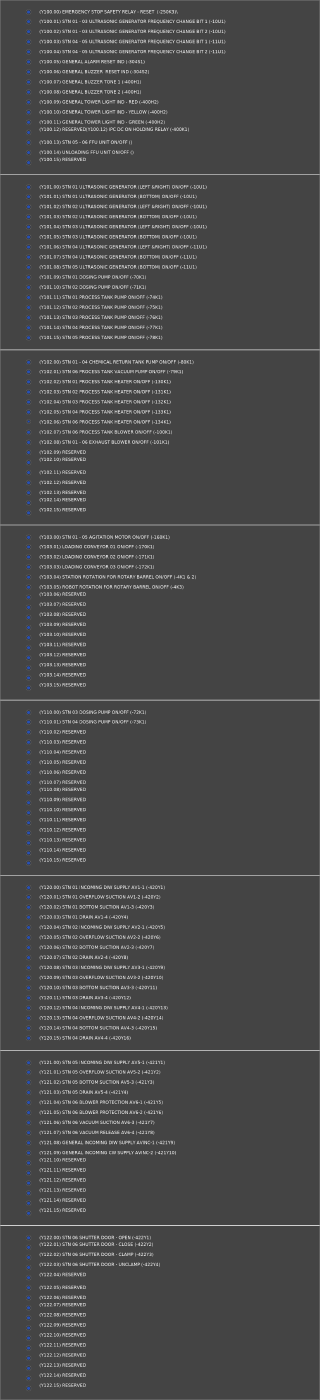
VISUALIZATION Popup_IOoutput  // 733x3198
    Rectangle (0,0 733x398)
    Label (87,15 625x24), "(Y100.00) EMERGENCY STOP SAFETY RELAY - RESET (-250K3)\"
    Label (87,37 625x24), "(Y100.01) STN 01 - 03 ULTRASONIC GENERATOR FREQUENCY CHANGE BIT 1 (-10U1)"
    Label (87,83 625x24), "(Y100.03) STN 04 - 05 ULTRASONIC GENERATOR FREQUENCY CHANGE BIT 1 (-11U1)"
    Label (87,60 625x24), "(Y100.02) STN 01 - 03 ULTRASONIC GENERATOR FREQUENCY CHANGE BIT 2 (-10U1)"
    Label (87,175 625x24), "(Y100.07) GENERAL BUZZER TONE 1 (-400H1)"
    Label (87,106 625x24), "(Y100.04) STN 04 - 05 ULTRASONIC GENERATOR FREQUENCY CHANGE BIT 2 (-11U1)"
    Label (87,129 625x24), "(Y100.05) GENERAL ALARM RESET IND (-304S1)"
    Label (87,152 625x24), "(Y100.06) GENERAL BUZZER RESET IND (-304S2)"
    Label (87,359 625x24), "(Y100.15) RESERVED"
    Label (87,198 625x24), "(Y100.08) GENERAL BUZZER TONE 2 (-400H1)"
    Label (87,221 625x24), "(Y100.09) GENERAL TOWER LIGHT IND - RED (-400H2)"
    Label (87,267 625x24), "(Y100.11) GENERAL TOWER LIGHT IND - GREEN (-400H2)"
    Label (87,244 625x24), "(Y100.10) GENERAL TOWER LIGHT IND - YELLOW (-400H2)"
    Label (87,290 625x24), "(Y100.12) RESERVED(Y100.12) IPC DC ON HOLDING RELAY (-400K1)"
    Label (87,313 625x24), "(Y100.13) STN 05 - 06 FFU UNIT ON/OFF ()"
    Label (87,336 625x24), "(Y100.14) UNLOADING FFU UNIT ON/OFF ()"
    Rectangle (0,400 733x398)
    Label (87,415 625x24), "(Y101.00) STN 01 ULTRASONIC GENERATOR (LEFT &RIGHT) ON/OFF (-10U1)"
    Label (87,437 625x24), "(Y101.01) STN 01 ULTRASONIC GENERATOR (BOTTOM) ON/OFF (-10U1)"
    Label (87,483 625x24), "(Y101.03) STN 02 ULTRASONIC GENERATOR (BOTTOM) ON/OFF (-10U1)"
    Label (87,460 625x24), "(Y101.02) STN 02 ULTRASONIC GENERATOR (LEFT &RIGHT) ON/OFF (-10U1)"
    Label (87,575 625x24), "(Y101.07) STN 04 ULTRASONIC GENERATOR (BOTTOM) ON/OFF (-11U1)"
    Label (87,506 625x24), "(Y101.04) STN 03 ULTRASONIC GENERATOR (LEFT &RIGHT) ON/OFF (-10U1)"
    Label (87,529 625x24), "(Y101.05) STN 03 ULTRASONIC GENERATOR (BOTTOM) ON/OFF (-10U1)"
    Label (87,552 625x24), "(Y101.06) STN 04 ULTRASONIC GENERATOR (LEFT &RIGHT) ON/OFF (-11U1)"
    Label (87,759 625x24), "(Y101.15) STN 05 PROCESS TANK PUMP ON/OFF (-78K1)"
    Label (87,598 625x24), "(Y101.08) STN 05 ULTRASONIC GENERATOR (BOTTOM) ON/OFF (-11U1)"
    Label (87,621 625x24), "(Y101.09) STN 01 DOSING PUMP ON/OFF (-70K1)"
    Label (87,667 625x24), "(Y101.11) STN 01 PROCESS TANK PUMP ON/OFF (-74K1)"
    Label (87,644 625x24), "(Y101.10) STN 02 DOSING PUMP ON/OFF (-71K1)"
    Label (87,690 625x24), "(Y101.12) STN 02 PROCESS TANK PUMP ON/OFF (-75K1)"
    Label (87,713 625x24), "(Y101.13) STN 03 PROCESS TANK PUMP ON/OFF (-76K1)"
    Label (87,736 625x24), "(Y101.14) STN 04 PROCESS TANK PUMP ON/OFF (-77K1)"
    Rectangle (0,800 733x398)
    Label (87,815 625x24), "(Y102.00) STN 01 - 04 CHEMICAL RETURN TANK PUMP ON/OFF (-80K1)"
    Label (87,837 625x24), "(Y102.01) STN 06 PROCESS TANK VACUUM PUMP ON/OFF (-79K1)"
    Label (87,883 625x24), "(Y102.03) STN 02 PROCESS TANK HEATER ON/OFF (-131K1)"
    Label (87,860 625x24), "(Y102.02) STN 01 PROCESS TANK HEATER ON/OFF (-130K1)"
    Label (87,975 625x24), "(Y102.07) STN 06 PROCESS TANK BLOWER ON/OFF (-100K1)"
    Label (87,906 625x24), "(Y102.04) STN 03 PROCESS TANK HEATER ON/OFF (-132K1)"
    Label (87,929 625x24), "(Y102.05) STN 04 PROCESS TANK HEATER ON/OFF (-133K1)"
    Label (87,952 625x24), "(Y102.06) STN 06 PROCESS TANK HEATER ON/OFF (-134K1)"
    Label (87,1159 625x24), "(Y102.15) RESERVED"
    Label (87,998 625x24), "(Y102.08) STN 01 - 06 EXHAUST BLOWER ON/OFF (-101K1)"
    Label (87,1021 625x24), "(Y102.09) RESERVED"
    Label (87,1067 625x24), "(Y102.11) RESERVED"
    Label (87,1044 625x24), "(Y102.10) RESERVED"
    Label (87,1090 625x24), "(Y102.12) RESERVED"
    Label (87,1113 625x24), "(Y102.13) RESERVED"
    Label (87,1136 625x24), "(Y102.14) RESERVED"
    Rectangle (0,1600 733x398)
    Label (87,1615 625x24), "(Y110.00) STN 03 DOSING PUMP ON/OFF (-72K1)"
    Label (87,1637 625x24), "(Y110.01) STN 04 DOSING PUMP ON/OFF (-73K1)"
    Label (87,1683 625x24), "(Y110.03) RESERVED"
    Label (87,1660 625x24), "(Y110.02) RESERVED"
    Label (87,1775 625x24), "(Y110.07) RESERVED"
    Label (87,1706 625x24), "(Y110.04) RESERVED"
    Label (87,1729 625x24), "(Y110.05) RESERVED"
    Label (87,1752 625x24), "(Y110.06) RESERVED"
    Label (87,1959 625x24), "(Y110.15) RESERVED"
    Label (87,1798 625x24), "(Y110.08) RESERVED"
    Label (87,1821 625x24), "(Y110.09) RESERVED"
    Label (87,1867 625x24), "(Y110.11) RESERVED"
    Label (87,1844 625x24), "(Y110.10) RESERVED"
    Label (87,1890 625x24), "(Y110.12) RESERVED"
    Label (87,1913 625x24), "(Y110.13) RESERVED"
    Label (87,1936 625x24), "(Y110.14) RESERVED"
    Rectangle (0,1200 733x398)
    Label (87,1215 625x24), "(Y103.00) STN 01 - 05 AGITATION MOTOR ON/OFF (-160K1)"
    Label (87,1237 625x24), "(Y103.01) LOADING CONVEYOR 01 ON/OFF (-170K1)"
    Label (87,1283 625x24), "(Y103.03) LOADING CONVEYOR 03 ON/OFF (-172K1)"
    Label (87,1260 625x24), "(Y103.02) LOADING CONVEYOR 02 ON/OFF (-171K1)"
    Label (87,1375 625x24), "(Y103.07) RESERVED"
    Label (87,1306 625x24), "(Y103.04) STATION ROTATION FOR ROTARY BARREL ON/OFF (-4K1 & 2)"
    Label (87,1329 625x24), "(Y103.05) ROBOT ROTATION FOR ROTARY BARREL ON/OFF (-4K3)"
    Label (87,1352 625x24), "(Y103.06) RESERVED"
    Label (87,1559 625x24), "(Y103.15) RESERVED"
    Label (87,1398 625x24), "(Y103.08) RESERVED"
    Label (87,1421 625x24), "(Y103.09) RESERVED"
    Label (87,1467 625x24), "(Y103.11) RESERVED"
    Label (87,1444 625x24), "(Y103.10) RESERVED"
    Label (87,1490 625x24), "(Y103.12) RESERVED"
    Label (87,1513 625x24), "(Y103.13) RESERVED"
    Label (87,1536 625x24), "(Y103.14) RESERVED"
    Rectangle (0,2000 733x398)
    Label (87,2015 625x24), "(Y120.00) STN 01 INCOMING DIW SUPPLY AV1-1 (-420Y1)"
    Label (87,2037 625x24), "(Y120.01) STN 01 OVERFLOW SUCTION AV1-2 (-420Y2)"
    Label (87,2083 625x24), "(Y120.03) STN 01 DRAIN AV1-4 (-420Y4)"
    Label (87,2060 625x24), "(Y120.02) STN 01 BOTTOM SUCTION AV1-3 (-420Y3)"
    Label (87,2175 625x24), "(Y120.07) STN 02 DRAIN AV2-4 (-420Y8)"
    Label (87,2106 625x24), "(Y120.04) STN 02 INCOMING DIW SUPPLY AV2-1 (-420Y5)"
    Label (87,2129 625x24), "(Y120.05) STN 02 OVERFLOW SUCTION AV2-2 (-420Y6)"
    Label (87,2152 625x24), "(Y120.06) STN 02 BOTTOM SUCTION AV2-3 (-420Y7)"
    Label (87,2359 625x24), "(Y120.15) STN 04 DRAIN AV4-4 (-420Y16)"
    Label (87,2198 625x24), "(Y120.08) STN 03 INCOMING DIW SUPPLY AV3-1 (-420Y9)"
    Label (87,2221 625x24), "(Y120.09) STN 03 OVERFLOW SUCTION AV3-2 (-420Y10)"
    Label (87,2267 625x24), "(Y120.11) STN 03 DRAIN AV3-4 (-420Y12)"
    Label (87,2244 625x24), "(Y120.10) STN 03 BOTTOM SUCTION AV3-3 (-420Y11)"
    Label (87,2290 625x24), "(Y120.12) STN 04 INCOMING DIW SUPPLY AV4-1 (-420Y13)"
    Label (87,2313 625x24), "(Y120.13) STN 04 OVERFLOW SUCTION AV4-2 (-420Y14)"
    Label (87,2336 625x24), "(Y120.14) STN 04 BOTTOM SUCTION AV4-3 (-420Y15)"
    Rectangle (0,2400 733x398)
    Label (87,2415 625x24), "(Y121.00) STN 05 INCOMING DIW SUPPLY AV5-1 (-421Y1)"
    Label (87,2437 625x24), "(Y121.01) STN 05 OVERFLOW SUCTION AV5-2 (-421Y2)"
    Label (87,2483 625x24), "(Y121.03) STN 05 DRAIN AV5-4 (-421Y4)"
    Label (87,2460 625x24), "(Y121.02) STN 05 BOTTOM SUCTION AV5-3 (-421Y3)"
    Label (87,2575 625x24), "(Y121.07) STN 06 VACUUM RELEASE AV6-4 (-421Y8)"
    Label (87,2506 625x24), "(Y121.04) STN 06 BLOWER PROTECTION AV6-1 (-421Y5)"
    Label (87,2529 625x24), "(Y121.05) STN 06 BLOWER PROTECTION AV6-2 (-421Y6)"
    Label (87,2552 625x24), "(Y121.06) STN 06 VACUUM SUCTION AV6-3 (-421Y7)"
    Label (87,2759 625x24), "(Y121.15) RESERVED"
    Label (87,2598 625x24), "(Y121.08) GENERAL INCOMING DIW SUPPLY AVINC-1 (-421Y9)"
    Label (87,2621 625x24), "(Y121.09) GENERAL INCOMING CW SUPPLY AVINC-2 (-421Y10)"
    Label (87,2667 625x24), "(Y121.11) RESERVED"
    Label (87,2644 625x24), "(Y121.10) RESERVED"
    Label (87,2690 625x24), "(Y121.12) RESERVED"
    Label (87,2713 625x24), "(Y121.13) RESERVED"
    Label (87,2736 625x24), "(Y121.14) RESERVED"
    Rectangle (0,2800 733x398)
    Label (87,2815 625x24), "(Y122.00) STN 06 SHUTTER DOOR - OPEN (-422Y1)"
    Label (87,2837 625x24), "(Y122.01) STN 06 SHUTTER DOOR - CLOSE (-422Y2)"
    Label (87,2883 625x24), "(Y122.03) STN 06 SHUTTER DOOR - UNCLAMP (-422Y4)"
    Label (87,2860 625x24), "(Y122.02) STN 06 SHUTTER DOOR - CLAMP (-422Y3)"
    Label (87,2975 625x24), "(Y122.07) RESERVED"
    Label (87,2906 625x24), "(Y122.04) RESERVED"
    Label (87,2929 625x24), "(Y122.05) RESERVED"
    Label (87,2952 625x24), "(Y122.06) RESERVED"
    Label (87,3159 625x24), "(Y122.15) RESERVED"
    Label (87,2998 625x24), "(Y122.08) RESERVED"
    Label (87,3021 625x24), "(Y122.09) RESERVED"
    Label (87,3067 625x24), "(Y122.11) RESERVED"
    Label (87,3044 625x24), "(Y122.10) RESERVED"
    Label (87,3090 625x24), "(Y122.12) RESERVED"
    Label (87,3113 625x24), "(Y122.13) RESERVED"
    Label (87,3136 625x24), "(Y122.14) RESERVED"
    Lamp1 (58,20 15x15), variable: ARbDO[eY10000_EmergencyStopSafetyRelay_Reset], style: Lamp-Lamp1-Blue
    Lamp1 (58,42 15x15), variable: ARbDO[eY10001_Stn01_03UltrasonicGeneratorFrequencyChangeBit1], style: Lamp-Lamp1-Blue
    Lamp1 (58,88 15x15), variable: ARbDO[eY10004_Stn04_05UltrasonicGeneratorFrequencyChangeBit2], style: Lamp-Lamp1-Blue
    Lamp1 (58,65 15x15), variable: ARbDO[eY10002_Stn01_03UltrasonicGeneratorFrequencyChangeBit2], style: Lamp-Lamp1-Blue
    Lamp1 (58,180 15x15), variable: ARbDO[eY10007_GeneralBuzzerTone1], style: Lamp-Lamp1-Blue
    Lamp1 (58,111 15x15), variable: ARbDI[eX10004_Stn02UltrasonicGeneratorBottom_Alarm], style: Lamp-Lamp1-Blue
    Lamp1 (58,134 15x15), variable: ARbDO[eY10005_GeneralAlarmResetInd], style: Lamp-Lamp1-Blue
    Lamp1 (58,157 15x15), variable: ARbDO[eY10006_GeneralBuzzerResetInd], style: Lamp-Lamp1-Blue
    Lamp1 (58,364 15x15), variable: ARbDO[eY10015_Reserved], style: Lamp-Lamp1-Blue
    Lamp1 (58,203 15x15), variable: ARbDO[eY10008_GeneralBuzzerTone2], style: Lamp-Lamp1-Blue
    Lamp1 (58,226 15x15), variable: ARbDO[eY10009_GeneralTowerLightInd_Red], style: Lamp-Lamp1-Blue
    Lamp1 (58,272 15x15), variable: ARbDO[eY10011_GeneralTowerLightInd_Green], style: Lamp-Lamp1-Blue
    Lamp1 (58,249 15x15), variable: ARbDO[eY10010_GeneralTowerLightInd_Yellow], style: Lamp-Lamp1-Blue
    Lamp1 (58,295 15x15), variable: ARbDO[eY10012_IpcDcOnHoldingRelay], style: Lamp-Lamp1-Blue
    Lamp1 (58,318 15x15), variable: ARbDO[eY10013_Stn05_06FfuUnitOnOff], style: Lamp-Lamp1-Blue
    Lamp1 (58,341 15x15), variable: ARbDO[eY10014_UnloadingFfuUnitOnOff], style: Lamp-Lamp1-Blue
    Lamp1 (58,420 15x15), variable: ARbDO[eY10100_Stn01UltrasonicGeneratorLeftRightOnOff], style: Lamp-Lamp1-Blue
    Lamp1 (58,442 15x15), variable: ARbDO[eY10101_Stn01UltrasonicGeneratorBottomOnOff], style: Lamp-Lamp1-Blue
    Lamp1 (58,488 15x15), variable: ARbDO[eY10103_Stn02UltrasonicGeneratorBottomOnOff], style: Lamp-Lamp1-Blue
    Lamp1 (58,465 15x15), variable: ARbDO[eY10102_Stn02UltrasonicGeneratorLeftRightOnOff], style: Lamp-Lamp1-Blue
    Lamp1 (58,580 15x15), variable: ARbDO[eY10107_Stn04UltrasonicGeneratorBottomOnOff], style: Lamp-Lamp1-Blue
    Lamp1 (58,511 15x15), variable: ARbDO[eY10104_Stn03UltrasonicGeneratorLeftRightOnOff], style: Lamp-Lamp1-Blue
    Lamp1 (58,534 15x15), variable: ARbDO[eY10105_Stn03UltrasonicGeneratorBottomOnOff], style: Lamp-Lamp1-Blue
    Lamp1 (58,557 15x15), variable: ARbDO[eY10106_Stn04UltrasonicGeneratorLeftRightOnOff], style: Lamp-Lamp1-Blue
    Lamp1 (58,764 15x15), variable: ARbDO[eY10115_Stn05ProcessTankPumpOnOff], style: Lamp-Lamp1-Blue
    Lamp1 (58,603 15x15), variable: ARbDO[eY10108_Stn05UltrasonicGeneratorBottomOnOff], style: Lamp-Lamp1-Blue
    Lamp1 (58,626 15x15), variable: ARbDO[eY10109_Stn01DosingPumpOnOff], style: Lamp-Lamp1-Blue
    Lamp1 (58,672 15x15), variable: ARbDO[eY10111_Stn01ProcessTankPumpOnOff], style: Lamp-Lamp1-Blue
    Lamp1 (58,649 15x15), variable: ARbDO[eY10110_Stn02DosingPumpOnOff], style: Lamp-Lamp1-Blue
    Lamp1 (58,695 15x15), variable: ARbDO[eY10112_Stn02ProcessTankPumpOnOff], style: Lamp-Lamp1-Blue
    Lamp1 (58,718 15x15), variable: ARbDO[eY10113_Stn03ProcessTankPumpOnOff], style: Lamp-Lamp1-Blue
    Lamp1 (58,741 15x15), variable: ARbDO[eY10114_Stn04ProcessTankPumpOnOff], style: Lamp-Lamp1-Blue
    Lamp1 (58,820 15x15), variable: ARbDO[eY10200_Stn01_04ChemicalReturnTankPumpOnOff], style: Lamp-Lamp1-Blue
    Lamp1 (58,842 15x15), variable: ARbDO[eY10201_Stn06ProcessTankVacuumPumpOnOff], style: Lamp-Lamp1-Blue
    Lamp1 (58,888 15x15), variable: ARbDO[eY10203_Stn02ProcessTankHeaterOnOff], style: Lamp-Lamp1-Blue
    Lamp1 (58,865 15x15), variable: ARbDO[eY10202_Stn01ProcessTankHeaterOnOff], style: Lamp-Lamp1-Blue
    Lamp1 (58,980 15x15), variable: ARbDO[eY10207_Stn06ProcessTankBlowerOnOff], style: Lamp-Lamp1-Blue
    Lamp1 (58,911 15x15), variable: ARbDI[eX10204_Stn05ProcessTankPumpMms_Tor_Trip], style: Lamp-Lamp1-Blue
    Lamp1 (58,934 15x15), variable: ARbDO[eY10205_Stn04ProcessTankHeaterOnOff], style: Lamp-Lamp1-Blue
    Lamp1 (58,957 15x12), variable: ARbDO[eY10206_Stn06ProcessTankHeaterOnOff], style: Lamp-Lamp1-Blue
    Lamp1 (58,1164 15x15), variable: ARbDO[eY10215_Reserved], style: Lamp-Lamp1-Blue
    Lamp1 (58,1003 15x15), variable: ARbDO[eY10208_Stn01_06ExhaustBlowerOnOff], style: Lamp-Lamp1-Blue
    Lamp1 (58,1026 15x15), variable: ARbDO[eY10209_Reserved], style: Lamp-Lamp1-Blue
    Lamp1 (58,1072 15x15), variable: ARbDO[eY10211_Reserved], style: Lamp-Lamp1-Blue
    Lamp1 (58,1049 15x15), variable: ARbDO[eY10210_Reserved], style: Lamp-Lamp1-Blue
    Lamp1 (58,1095 15x15), variable: ARbDO[eY10212_Reserved], style: Lamp-Lamp1-Blue
    Lamp1 (58,1118 15x15), variable: ARbDO[eY10213_Reserved], style: Lamp-Lamp1-Blue
    Lamp1 (58,1141 15x15), variable: ARbDO[eY10214_Reserved], style: Lamp-Lamp1-Blue
    Lamp1 (58,1620 15x15), variable: ARbDO[eY11000_Stn03DosingPumpOnOff], style: Lamp-Lamp1-Blue
    Lamp1 (58,1642 15x15), variable: ARbDO[eY11001_Stn04DosingPumpOnOff], style: Lamp-Lamp1-Blue
    Lamp1 (58,1688 15x15), variable: ARbDO[eY11003_Reserved], style: Lamp-Lamp1-Blue
    Lamp1 (58,1665 15x15), variable: ARbDO[eY11002_Reserved], style: Lamp-Lamp1-Blue
    Lamp1 (58,1780 15x15), variable: ARbDO[eY11007_Reserved], style: Lamp-Lamp1-Blue
    Lamp1 (58,1711 15x15), variable: ARbDO[eY11004_Reserved], style: Lamp-Lamp1-Blue
    Lamp1 (58,1734 15x15), variable: ARbDO[eY11005_Reserved], style: Lamp-Lamp1-Blue
    Lamp1 (58,1757 15x15), variable: ARbDO[eY11006_Reserved], style: Lamp-Lamp1-Blue
    Lamp1 (58,1964 15x15), variable: ARbDO[eY11015_Reserved], style: Lamp-Lamp1-Blue
    Lamp1 (58,1803 15x15), variable: ARbDO[eY11008_Reserved], style: Lamp-Lamp1-Blue
    Lamp1 (58,1826 15x15), variable: ARbDO[eY11009_Reserved], style: Lamp-Lamp1-Blue
    Lamp1 (58,1872 15x15), variable: ARbDO[eY11011_Reserved], style: Lamp-Lamp1-Blue
    Lamp1 (58,1849 15x15), variable: ARbDI[eX10410_Structure01DripPanSensor_Leak], style: Lamp-Lamp1-Blue
    Lamp1 (58,1895 15x15), variable: ARbDO[eY11012_Reserved], style: Lamp-Lamp1-Blue
    Lamp1 (58,1918 15x15), variable: ARbDO[eY11013_Reserved], style: Lamp-Lamp1-Blue
    Lamp1 (58,1941 15x15), variable: ARbDO[eY11014_Reserved], style: Lamp-Lamp1-Blue
    Lamp1 (58,1220 15x15), variable: ARbDO[eY10300_Stn01_05AgitationMotorOnOff], style: Lamp-Lamp1-Blue
    Lamp1 (58,1242 15x15), variable: ARbDO[eY10301_LoadingConveyor01OnOff], style: Lamp-Lamp1-Blue
    Lamp1 (58,1288 15x15), variable: ARbDO[eY10303_LoadingConveyor03OnOff], style: Lamp-Lamp1-Blue
    Lamp1 (58,1265 15x15), variable: ARbDO[eY10302_LoadingConveyor02OnOff], style: Lamp-Lamp1-Blue
    Lamp1 (58,1380 15x15), variable: ARbDO[eY10307_Reserved], style: Lamp-Lamp1-Blue
    Lamp1 (58,1311 15x15), variable: ARbDO[eY10304_StationRotationForRotaryBarrelOnOff], style: Lamp-Lamp1-Blue
    Lamp1 (58,1334 15x15), variable: ARbDO[eY10305_RobotRotationForRotaryBarrelOnOff], style: Lamp-Lamp1-Blue
    Lamp1 (58,1357 15x15), variable: ARbDO[eY10306_Reserved], style: Lamp-Lamp1-Blue
    Lamp1 (58,1564 15x15), variable: ARbDO[eY10315_Reserved], style: Lamp-Lamp1-Blue
    Lamp1 (58,1403 15x15), variable: ARbDO[eY10308_Reserved], style: Lamp-Lamp1-Blue
    Lamp1 (58,1426 15x15), variable: ARbDO[eY10309_Reserved], style: Lamp-Lamp1-Blue
    Lamp1 (58,1472 15x15), variable: ARbDO[eY10311_Reserved], style: Lamp-Lamp1-Blue
    Lamp1 (58,1449 15x15), variable: ARbDO[eY10310_Reserved], style: Lamp-Lamp1-Blue
    Lamp1 (58,1495 15x15), variable: ARbDO[eY10312_Reserved], style: Lamp-Lamp1-Blue
    Lamp1 (58,1518 15x15), variable: ARbDO[eY10313_Reserved], style: Lamp-Lamp1-Blue
    Lamp1 (58,1541 15x15), variable: ARbDO[eY10314_Reserved], style: Lamp-Lamp1-Blue
    Lamp1 (58,2020 15x15), variable: ARbDO[eY12000_Stn01IncomingDiwSupplyAv1_1], style: Lamp-Lamp1-Blue
    Lamp1 (58,2042 15x15), variable: ARbDO[eY12001_Stn01OverflowSuctionAv1_2], style: Lamp-Lamp1-Blue
    Lamp1 (58,2088 15x15), variable: ARbDO[eY12003_Stn01DrainAv1_4], style: Lamp-Lamp1-Blue
    Lamp1 (58,2065 15x15), variable: ARbDO[eY12002_Stn01BottomSuctionAv1_3], style: Lamp-Lamp1-Blue
    Lamp1 (58,2180 15x15), variable: ARbDO[eY12007_Stn02DrainAv2_4], style: Lamp-Lamp1-Blue
    Lamp1 (58,2111 15x15), variable: ARbDO[eY12004_Stn02IncomingDiwSupplyAv2_1], style: Lamp-Lamp1-Blue
    Lamp1 (58,2134 15x15), variable: ARbDO[eY12005_Stn02OverflowSuctionAv2_2], style: Lamp-Lamp1-Blue
    Lamp1 (58,2157 15x15), variable: ARbDO[eY12006_Stn02BottomSuctionAv2_3], style: Lamp-Lamp1-Blue
    Lamp1 (58,2364 15x15), variable: ARbDO[eY12015_Stn04DrainAv4_4], style: Lamp-Lamp1-Blue
    Lamp1 (58,2203 15x15), variable: ARbDO[eY12008_Stn03IncomingDiwSupplyAv3_1], style: Lamp-Lamp1-Blue
    Lamp1 (58,2226 15x15), variable: ARbDO[eY12009_Stn03OverflowSuctionAv3_2], style: Lamp-Lamp1-Blue
    Lamp1 (58,2272 15x15), variable: ARbDO[eY12011_Stn03DrainAv3_4], style: Lamp-Lamp1-Blue
    Lamp1 (58,2249 15x15), variable: ARbDO[eY12010_Stn03BottomSuctionAv3_3], style: Lamp-Lamp1-Blue
    Lamp1 (58,2295 15x15), variable: ARbDO[eY12012_Stn04IncomingDiwSupplyAv4_1], style: Lamp-Lamp1-Blue
    Lamp1 (58,2318 15x15), variable: ARbDO[eY12013_Stn04OverflowSuctionAv4_2], style: Lamp-Lamp1-Blue
    Lamp1 (58,2341 15x15), variable: ARbDO[eY12014_Stn04BottomSuctionAv4_3], style: Lamp-Lamp1-Blue
    Lamp1 (58,2420 15x15), variable: ARbDO[eY12100_Stn05IncomingDiwSupplyAv5_1], style: Lamp-Lamp1-Blue
    Lamp1 (58,2442 15x15), variable: ARbDO[eY12101_Stn05IncomingCwSupplyAv5_2], style: Lamp-Lamp1-Blue
    Lamp1 (58,2488 15x15), variable: ARbDO[eY12103_Stn05DrainAv5_4], style: Lamp-Lamp1-Blue
    Lamp1 (58,2465 15x15), variable: ARbDO[eY12102_Stn05BottomSuctionAv5_3], style: Lamp-Lamp1-Blue
    Lamp1 (58,2580 15x15), variable: ARbDO[eY12107_Stn06VacuumReleaseAv6_4], style: Lamp-Lamp1-Blue
    Lamp1 (58,2511 15x15), variable: ARbDO[eY12104_Stn06BlowerProtectionAv6_1], style: Lamp-Lamp1-Blue
    Lamp1 (58,2534 15x15), variable: ARbDO[eY12105_Stn06BlowerProtectionAv6_2], style: Lamp-Lamp1-Blue
    Lamp1 (58,2557 15x15), variable: ARbDO[eY12106_Stn06VacuumSuctionAv6_3], style: Lamp-Lamp1-Blue
    Lamp1 (58,2764 15x15), variable: ARbDO[eY12115_Reserved], style: Lamp-Lamp1-Blue
    Lamp1 (58,2603 15x15), variable: ARbDO[eY12108_GeneralIncomingDiwSupplyAvinc_1], style: Lamp-Lamp1-Blue
    Lamp1 (58,2626 15x15), variable: ARbDO[eY12109_GeneralIncomingCwSupplyAvinc_2], style: Lamp-Lamp1-Blue
    Lamp1 (58,2672 15x15), variable: ARbDO[eY12111_Reserved], style: Lamp-Lamp1-Blue
    Lamp1 (58,2649 15x15), variable: ARbDO[eY12110_Reserved], style: Lamp-Lamp1-Blue
    Lamp1 (58,2695 15x15), variable: ARbDO[eY12112_Reserved], style: Lamp-Lamp1-Blue
    Lamp1 (58,2718 15x15), variable: ARbDO[eY12113_Reserved], style: Lamp-Lamp1-Blue
    Lamp1 (58,2741 15x15), variable: ARbDO[eY12114_Reserved], style: Lamp-Lamp1-Blue
    Lamp1 (58,2820 15x15), variable: ARbDO[eY12200_Stn06SlidingDoor_Open], style: Lamp-Lamp1-Blue
    Lamp1 (58,2842 15x15), variable: ARbDO[eY12201_Stn06SlidingDoor_Close], style: Lamp-Lamp1-Blue
    Lamp1 (58,2888 15x15), variable: ARbDO[eY12203_Stn06SlidingDoor_Unclamp], style: Lamp-Lamp1-Blue
    Lamp1 (58,2865 15x15), variable: ARbDO[eY12202_Stn06SlidingDoor_Clamp], style: Lamp-Lamp1-Blue
    Lamp1 (58,2980 15x15), variable: ARbDO[eY12207_Reserved], style: Lamp-Lamp1-Blue
    Lamp1 (58,2911 15x15), variable: ARbDO[eY12204_Reserved], style: Lamp-Lamp1-Blue
    Lamp1 (58,2934 15x15), variable: ARbDO[eY12205_Reserved], style: Lamp-Lamp1-Blue
    Lamp1 (58,2957 15x15), variable: ARbDO[eY12206_Reserved], style: Lamp-Lamp1-Blue
    Lamp1 (58,3164 15x15), variable: ARbDO[eY12215_Reserved], style: Lamp-Lamp1-Blue
    Lamp1 (58,3003 15x15), variable: ARbDO[eY12208_Reserved], style: Lamp-Lamp1-Blue
    Lamp1 (58,3026 15x15), variable: ARbDO[eY12210_Reserved], style: Lamp-Lamp1-Blue
    Lamp1 (58,3072 15x15), variable: ARbDO[eY12211_Reserved], style: Lamp-Lamp1-Blue
    Lamp1 (58,3049 15x15), variable: ARbDO[eY12210_Reserved], style: Lamp-Lamp1-Blue
    Lamp1 (58,3095 15x15), variable: ARbDO[eY12212_Reserved], style: Lamp-Lamp1-Blue
    Lamp1 (58,3118 15x15), variable: ARbDO[eY12213_Reserved], style: Lamp-Lamp1-Blue
    Lamp1 (58,3141 15x15), variable: ARbDO[eY12214_Reserved], style: Lamp-Lamp1-Blue
END_VISUALIZATION

(* stored: Version 1.1.0.1, ProductVersion 3.1.4024.12
   Visu Popup_IOoutput: Id {d20d2f26-0d00-41bd-9964-034fcaa3c414} *)
